// TwinCAT 3 PLC project tcl_AdsObjects
// Title: tcl_AdsObjects
// Company: Red Rock Controls Limited
// Author: R Christopher
// ProjectVersion: 1.1.4.0
// Description: Wrapper classes for Ads function blocks
// ProgramVersion: 3.1.4022.0
// libraries:
//   Tc2_Standard, * (Beckhoff Automation GmbH)
//   Tc2_System, * (Beckhoff Automation GmbH)
//   Tc2_Utilities, * (Beckhoff Automation GmbH)
//   Tc3_Module, * (Beckhoff Automation GmbH)
//   tcl_BaseClasses, * (Red Rock Controls Limited)
//   tcl_UnitTestLibrary, * (Red Rock Controls Limited)
// project tree:
//   / GlobalTextList.TcGTLO
//   POUs/Classes/By Index Group/ T_AdsRead.TcPOU, T_AdsReadWrite.TcPOU, T_AdsWrite.TcPOU
//   POUs/Classes/By Symbol Name/ T_AdsReadBySymbolName.TcPOU, T_AdsReadWriteBySymbolName.TcPOU, T_AdsWriteBySymbolName.TcPOU
//   POUs/Classes/Info/ ST_RawSymbolInfo.TcDUT, T_AdsReadSymbolName.TcPOU, T_AdsReadSymbolInfoByName.TcPOU
//   POUs/Classes/On Change/StructureMonitor/ T_StructureMonitor.TcPOU
//   POUs/Classes/On Change/ T_AdsWriteOnChange.TcPOU
//   Tasks/ PlcTask.TcTTO
//   UnitTests/RPC Example Class/ T_Integer.TcPOU
//   UnitTests/ PB_TestRunner.TcPOU, TestSuite_AdsTests.TcPOU, Test_ReadBySymbolName.TcPOU, Test_ReadBySymbolInfoByName.TcPOU, Test_ReadByIndexGroupAndOffset.TcPOU, Test_ReadSymbolName.TcPOU, Test_ReadBySymbolName_KeepingHandle.TcPOU, Test_ReadWriteBySymbolName.TcPOU, Test_ReadWriteBySymbolName_KeepingHandle.TcPOU, Test_WriteBySymbolName.TcPOU, Test_WriteBySymbolName_KeepingHandle.TcPOU
//   Version/ Global_Version.TcGVL
// real-time tasks:
//   TASK PlcTask: cycle T#10ms, priority 20, ADS port 350

CONFIGURATION tcl_AdsObjects
    RESOURCE PLC ON TwinCAT3
        TASK PlcTask(INTERVAL := T#10ms, PRIORITY := 20);
        PROGRAM PB_TestRunner WITH PlcTask : PB_TestRunner;
    END_RESOURCE
END_CONFIGURATION

// ---- POUs/Classes/Info/ST_RawSymbolInfo.TcDUT
TYPE
    INTERNAL ST_RawSymbolInfo :
    STRUCT
        Address : ULINT;
        Length  : ULINT;
    END_STRUCT
END_TYPE

// ---- Version/Global_Version.TcGVL
{attribute 'TcGenerated'}
{attribute 'no-analysis'}
{attribute 'linkalways'}
// This function has been automatically generated from the project information.
VAR_GLOBAL CONSTANT
	{attribute 'const_non_replaced'}
	stLibVersion_tcl_AdsObjects : ST_LibVersion := (iMajor := 1, iMinor := 1, iBuild := 4, iRevision := 0, nFlags := 1, sVersion := '1.1.4.0');
END_VAR

// ---- UnitTests/PB_TestRunner.TcPOU
PROGRAM PB_TestRunner
VAR
    TestSuite_AdsTests : TestSuite_AdsTests;
END_VAR

TestSuite_AdsTests();

END_PROGRAM

// ---- UnitTests/TestSuite_AdsTests.TcPOU
FUNCTION_BLOCK TestSuite_AdsTests
VAR
    TestRunner : T_TestRunner;
    // Inhibit unused variable warning...                                                        
    {attribute 'analysis' := '-33'} Test_ReadSymbolName                      : Test_ReadSymbolName(TestRunner);
    {attribute 'analysis' := '-33'} Test_ReadBySymbolName                    : Test_ReadBySymbolName(TestRunner);
    {attribute 'analysis' := '-33'} Test_ReadBySymbolName_KeepingHandle      : Test_ReadBySymbolName_KeepingHandle(TestRunner);
    {attribute 'analysis' := '-33'} Test_ReadWriteBySymbolName               : Test_ReadWriteBySymbolName(TestRunner);
    {attribute 'analysis' := '-33'} Test_ReadWriteBySymbolName_KeepingHandle : Test_ReadWriteBySymbolName_KeepingHandle(TestRunner);
    {attribute 'analysis' := '-33'} Test_WriteBySymbolName                   : Test_WriteBySymbolName(TestRunner);
    {attribute 'analysis' := '-33'} Test_WriteBySymbolName_KeepingHandle     : Test_WriteBySymbolName_KeepingHandle(TestRunner);
    {attribute 'analysis' := '-33'} Test_ReadBySymbolInfoByName              : Test_ReadBySymbolInfoByName(TestRunner);
    {attribute 'analysis' := '-33'} Test_ReadByIndexGroupAndOffset           : Test_ReadByIndexGroupAndOffset(TestRunner);

END_VAR

TestRunner(TestSuiteName := 'TestSuite_AdsTests');

END_FUNCTION_BLOCK

// ---- UnitTests/Test_ReadSymbolName.TcPOU
FUNCTION_BLOCK Test_ReadSymbolName EXTENDS T_UnitTestBase
VAR
    AdsPort                                                                                 : UINT;
    AdsReadSymbolName                                                                       : T_AdsReadSymbolName;
    SymbolWithAVeryVeryVeryVeryVeryVeryVeryVeryVeryVeryVeryVeryVeryVeryVeryVeryVeryLongName : INT;
    State                                                                                   : INT;
END_VAR

METHOD Init
State := 0;
END_METHOD

{attribute 'analysis' := '-33'} // inhibit unused variable warning
METHOD RunTest
VAR_OUTPUT
    TestCompleted : BOOL;
    TestFailed    : BOOL;
END_VAR
VAR_INST
    SymbolName : T_MaxString;
END_VAR
CASE State OF
    0:
        AdsPort := _AppInfo.AdsPort;
        AdsReadSymbolName.Execute(Address := ADR(SymbolWithAVeryVeryVeryVeryVeryVeryVeryVeryVeryVeryVeryVeryVeryVeryVeryVeryVeryLongName),
                                  Length  := SIZEOF(SymbolWithAVeryVeryVeryVeryVeryVeryVeryVeryVeryVeryVeryVeryVeryVeryVeryVeryVeryLongName),
                                  PlcPort := AdsPort);
        State := 10;

    10:
        IF NOT AdsReadSymbolName.Execution.Busy THEN
            SymbolName := AdsReadSymbolName.SymbolName;
            State      := 20;
        END_IF

    20:
        AssertTrue(Source    := TestName,
                   Condition := (SymbolName = 'PB_TestRunner.TestSuite_AdsTests.Test_ReadSymbolName.SymbolWithAVeryVeryVeryVeryVeryVeryVeryVeryVeryVeryVeryVeryVeryVeryVeryVeryVeryLongName'),
                   Message   := 'SymbolName read incorrectly',
                   Failed    => TestFailed);

        TestCompleted := TRUE;
END_CASE

AdsReadSymbolName();
END_METHOD

END_FUNCTION_BLOCK

// ---- POUs/Classes/Info/T_AdsReadSymbolName.TcPOU
FUNCTION_BLOCK T_AdsReadSymbolName
VAR
    _Execution    : T_Execution;
    _Address      : PVOID;
    _Length       : UDINT;
    _PlcPort      : UINT;
    _SymbolName   : T_MaxString;
    RawSymbolInfo : ST_RawSymbolInfo;
    AdsRdWrt1     : ADSRDWRTEX;
END_VAR
VAR CONSTANT
    PLCADS_IGR_SYMNAME_BY_ADDR_SIZE : UDINT := 16#40A1;
END_VAR

IF _Execution.Aborting THEN
    _Execution.SetAborted();
END_IF

IF _Execution.Starting THEN
    RawSymbolInfo.Address := _Address;
    RawSymbolInfo.Length  := _Length;
    MEMSET(ADR(_SymbolName), 0, SIZEOF(_SymbolName));
END_IF

AdsRdWrt1(NETID    :=,
          PORT     := _PlcPort,
          IDXGRP   := PLCADS_IGR_SYMNAME_BY_ADDR_SIZE,
          IDXOFFS  := 0,
          WRITELEN := SIZEOF(RawSymbolInfo),
          READLEN  := SIZEOF(SymbolName),
          SRCADDR  := ADR(RawSymbolInfo),
          DESTADDR := ADR(_SymbolName),
          WRTRD    := _Execution.Starting,
          TMOUT    := T#2s,
          BUSY     =>,
          ERR      =>,
          ERRID    =>,
          COUNT_R  =>);

IF _Execution.Starting THEN
    _Execution.SetBusy();
END_IF

IF _Execution.Busy AND NOT AdsRdWrt1.BUSY THEN
    IF AdsRdWrt1.ERR THEN
        _Execution.SetError(F_ErrorIdToString(AdsRdWrt1.ERRID));
    ELSE
        _Execution.SetDone();
    END_IF
END_IF

METHOD Execute : BOOL
VAR_INPUT
    Address : PVOID;
    Length  : UDINT;
    PlcPort : UINT;
END_VAR
THIS^._Address    := Address;
THIS^._Length     := Length;
THIS^._PlcPort    := PlcPort;
THIS^._SymbolName := '';
Execute           := THIS^._Execution.Start();
END_METHOD

PROPERTY Execution : I_Execution
GET
Execution := _Execution;
END_GET
END_PROPERTY

PROPERTY SymbolName : T_MaxString
GET
SymbolName := _SymbolName;
END_GET
END_PROPERTY

END_FUNCTION_BLOCK

// ---- UnitTests/Test_ReadBySymbolName.TcPOU
FUNCTION_BLOCK Test_ReadBySymbolName EXTENDS T_UnitTestBase
VAR
    AdsPort             : UINT;
    AdsReadBySymbolName : T_AdsReadBySymbolName;
    AdsReadSymbolName   : T_AdsReadSymbolName;
    ValueToRead         : INT;
    State               : INT;
END_VAR

METHOD Init
State := 0;
END_METHOD

{attribute 'analysis' := '-33'} // inhibit unused variable warning
METHOD RunTest
VAR_OUTPUT
    TestCompleted : BOOL;
    TestFailed    : BOOL;
END_VAR
VAR_INST
    SymbolName : T_MaxString;
    ReadResult : INT;
END_VAR
CASE State OF
    0:
        AdsPort     := _AppInfo.AdsPort;
        ValueToRead := 1234;
        ReadResult  := 0;
        AdsReadSymbolName.Execute(Address := ADR(ValueToRead),
                                  Length  := SIZEOF(ValueToRead),
                                  PlcPort := AdsPort);
        State := 10;

    10:
        IF NOT AdsReadSymbolName.Execution.Busy THEN
            SymbolName := AdsReadSymbolName.SymbolName;
            State      := 20;
        END_IF

    20:
        AdsReadBySymbolName.Execute(AmsNetId         := '',
                                    Port             := AdsPort,
                                    SymbolName       := SymbolName,
                                    ReadDataAddress  := ADR(ReadResult),
                                    ReadDataLength   := SIZEOF(ReadResult),
                                    KeepSymbolHandle := FALSE);

        State := 30;

    30:
        IF NOT AdsReadBySymbolName.Execution.Busy THEN
            State := 40;
        END_IF

    40:
        AssertTrue(Source    := TestName,
                   Condition := (ReadResult = 1234),
                   Message   := 'Read result <> 1234',
                   Failed    => TestFailed);

        TestCompleted := TRUE;
END_CASE

AdsReadBySymbolName();
AdsReadSymbolName();
END_METHOD

END_FUNCTION_BLOCK

// ---- POUs/Classes/By Symbol Name/T_AdsReadBySymbolName.TcPOU
FUNCTION_BLOCK T_AdsReadBySymbolName
VAR
    _Execution   : T_Execution;
    StateMonitor : T_ValueMonitor;
    State        : INT;

    AmsNetId         : T_AmsNetId;
    Port             : T_AmsPort;
    SymbolName       : T_MaxString;
    ReadDataAddress  : PVOID;
    ReadDataLength   : UDINT;
    KeepSymbolHandle : BOOL;
    SymbolHandle     : DWORD := 0;
    RetryCounter     : T_Counter;

    AdsReadWrite_GetSymHandle : T_AdsReadWrite;
    AdsRead_ReadFromSymbol    : T_AdsRead;
    AdsWrite_ReleaseSymHandle : T_AdsWrite;

END_VAR
VAR CONSTANT
    sInit          : INT := 0;
    sGetHandle     : INT := 1;
    sReadData      : INT := 2;
    sReleaseHandle : INT := 3;
END_VAR

IF _Execution.Aborting THEN
    State := sInit;
    _Execution.SetAborted();
END_IF

StateMonitor.Test(State);
CASE State OF
    sInit:
        IF _Execution.Starting THEN
            _Execution.SetBusy();
            RetryCounter.Reset();
            IF SymbolHandle = 0 THEN
                State := sGetHandle;
            ELSE
                State := sReadData;
            END_IF
        END_IF

    sGetHandle:
        IF StateMonitor.Changed THEN
            // Get a symbol handle from the runtime...
            AdsReadWrite_GetSymHandle.Execute(AmsNetId           := AmsNetId,
                                              Port               := Port,
                                              IndexGroup         := ADSIGRP_SYM_HNDBYNAME,
                                              IndexOffset        := 0,
                                              ArgsAddress        := ADR(SymbolName),
                                              ArgsLength         := INT_TO_UDINT(LEN(SymbolName)),
                                              ReturnValueAddress := ADR(SymbolHandle),
                                              ReturnValueLength  := SIZEOF(SymbolHandle));
        ELSE
            IF AdsReadWrite_GetSymHandle.Execution.Done THEN
                State := sReadData;
            END_IF
            IF AdsReadWrite_GetSymHandle.Execution.Error THEN
                _Execution.SetError(AdsReadWrite_GetSymHandle.Execution.ErrorMsg);
                SymbolHandle := 0;
                State        := sInit;
            END_IF
        END_IF

    sReadData:
        IF StateMonitor.Changed THEN
            // Read the data to from the symbol...
            AdsRead_ReadFromSymbol.Execute(AmsNetId    := AmsNetId,
                                           Port        := Port,
                                           IndexGroup  := ADSIGRP_SYM_VALBYHND,
                                           IndexOffset := SymbolHandle,
                                           DataLength  := ReadDataLength,
                                           DataAddress := ReadDataAddress);
        ELSE
            IF AdsRead_ReadFromSymbol.Execution.Done THEN
                IF KeepSymbolHandle THEN
                    _Execution.SetDone();
                    State := sInit;
                ELSE
                    State := sReleaseHandle;
                END_IF

            ELSIF AdsRead_ReadFromSymbol.Execution.Error THEN
                // Retry if it failed due to an online change invalidating the symbol handle...
                IF RetryCounter.Value = 0 THEN
                    RetryCounter.Inc();
                    SymbolHandle := 0;
                    State        := sGetHandle;
                ELSE
                    _Execution.SetError(AdsRead_ReadFromSymbol.Execution.ErrorMsg);
                    SymbolHandle := 0;
                    State        := sInit;
                END_IF
            END_IF
        END_IF

    sReleaseHandle:
        IF StateMonitor.Changed THEN
            // Release the symbol handle......
            AdsWrite_ReleaseSymHandle.Execute(AmsNetId    := AmsNetId,
                                              Port        := Port,
                                              IndexGroup  := ADSIGRP_SYM_RELEASEHND,
                                              IndexOffset := SymbolHandle,
                                              DataLength  := 0,
                                              DataAddress := 0);
        ELSE
            IF AdsWrite_ReleaseSymHandle.Execution.Done THEN
                // Handle write error to the symbol...
                IF AdsRead_ReadFromSymbol.Execution.Error THEN
                    _Execution.SetError(AdsRead_ReadFromSymbol.Execution.ErrorMsg);
                ELSE
                    _Execution.SetDone();
                END_IF
                SymbolHandle := 0;
                State        := sInit;
            ELSIF AdsWrite_ReleaseSymHandle.Execution.Error THEN
                // Handle release handle error...
                _Execution.SetError(AdsWrite_ReleaseSymHandle.Execution.ErrorMsg);
                SymbolHandle := 0;
                State        := sInit;
            END_IF
        END_IF

END_CASE

AdsReadWrite_GetSymHandle();
AdsRead_ReadFromSymbol();
AdsWrite_ReleaseSymHandle();

METHOD Execute : BOOL
VAR_INPUT
    AmsNetId         : T_AmsNetId;
    Port             : T_AmsPort;
    SymbolName       : T_MaxString;
    ReadDataAddress  : PVOID;
    ReadDataLength   : UDINT;
    KeepSymbolHandle : BOOL;
END_VAR
THIS^.AmsNetId         := AmsNetId;
THIS^.Port             := Port;
THIS^.SymbolName       := SymbolName;
THIS^.ReadDataAddress  := ReadDataAddress;
THIS^.ReadDataLength   := ReadDataLength;
THIS^.KeepSymbolHandle := KeepSymbolHandle;

Execute := _Execution.Start();
END_METHOD

PROPERTY Execution : I_Execution
GET
Execution := _Execution;
END_GET
END_PROPERTY

END_FUNCTION_BLOCK

// ---- POUs/Classes/By Index Group/T_AdsReadWrite.TcPOU
FUNCTION_BLOCK T_AdsReadWrite
VAR_INPUT
END_VAR
VAR_OUTPUT
END_VAR
VAR
    AdsReadWrite : ADSRDWRT;
    _Execution   : T_Execution;
END_VAR

IF _Execution.Aborting THEN
    _Execution.SetAborted();
END_IF

AdsReadWrite(NETID    :=,
             PORT     :=,
             IDXGRP   :=,
             IDXOFFS  :=,
             WRITELEN :=,
             READLEN  :=,
             SRCADDR  :=,
             DESTADDR :=,
             WRTRD    := _Execution.Starting,
             TMOUT    :=,
             BUSY     =>,
             ERR      =>,
             ERRID    =>);

IF _Execution.Starting THEN
    _Execution.SetBusy();
END_IF
IF _Execution.Busy AND NOT AdsReadWrite.BUSY THEN
    IF AdsReadWrite.ERR THEN
        _Execution.SetError(F_ErrorIdToString(AdsReadWrite.ERRID));
    ELSE
        _Execution.SetDone();
    END_IF
END_IF

METHOD Execute : BOOL
VAR_INPUT
    AmsNetId           : T_AmsNetID;
    Port               : T_AmsPort;
    IndexGroup         : UDINT;
    IndexOffset        : UDINT;
    ArgsAddress        : PVOID;
    ArgsLength         : UDINT;
    ReturnValueAddress : PVOID;
    ReturnValueLength  : UDINT;
END_VAR
IF _Execution.Start() THEN
    AdsReadWrite.NETID   := AmsNetId;
    AdsReadWrite.PORT    := Port;
    AdsReadWrite.IDXGRP  := IndexGroup;
    AdsReadWrite.IDXOFFS := IndexOffset;
    // Data to be written...
    AdsReadWrite.SRCADDR  := ArgsAddress;
    AdsReadWrite.WRITELEN := ArgsLength;
    // Data returned...
    AdsReadWrite.DESTADDR := ReturnValueAddress;
    AdsReadWrite.READLEN  := ReturnValueLength;
END_IF
END_METHOD

PROPERTY Execution : I_Execution
GET
Execution := _Execution;
END_GET
END_PROPERTY

END_FUNCTION_BLOCK

// ---- POUs/Classes/By Index Group/T_AdsRead.TcPOU
FUNCTION_BLOCK T_AdsRead
VAR
    _Execution : T_Execution;
    AdsRead1   : ADSREAD := (TMOUT := T#2S);
END_VAR

IF _Execution.Aborting THEN
    _Execution.SetAborted();
END_IF

AdsRead1(NETID    :=,
         PORT     :=,
         IDXGRP   :=,
         IDXOFFS  :=,
         LEN      :=,
         DESTADDR :=,
         READ     := _Execution.Starting,
         TMOUT    :=,
         BUSY     =>,
         ERR      =>,
         ERRID    =>);

IF _Execution.Starting THEN
    _Execution.SetBusy();
END_IF
IF _Execution.Busy AND NOT AdsRead1.BUSY THEN
    IF AdsRead1.ERR THEN
        _Execution.SetError(F_ErrorIdToString(AdsRead1.ERRID));
    ELSE
        _Execution.SetDone();
    END_IF
END_IF

METHOD Execute : BOOL
VAR_INPUT
    AmsNetId    : T_AmsNetid;
    Port        : T_AmsPort;
    IndexGroup  : UDINT;
    IndexOffset : UDINT;
    DataLength  : UDINT;
    DataAddress : PVOID;
END_VAR
AdsRead1.NETID    := AmsNetId;
AdsRead1.PORT     := Port;
AdsRead1.IDXGRP   := IndexGroup;
AdsRead1.IDXOFFS  := IndexOffset;
AdsRead1.LEN      := DataLength;
AdsRead1.DESTADDR := DataAddress;

Execute := _Execution.Start();
END_METHOD

PROPERTY Execution : I_Execution
GET
Execution := _Execution;
END_GET
END_PROPERTY

END_FUNCTION_BLOCK

// ---- POUs/Classes/By Index Group/T_AdsWrite.TcPOU
FUNCTION_BLOCK T_AdsWrite
VAR
    _Execution : T_Execution;
    AdsWrite1  : ADSWRITE := (TMOUT := T#2S);
END_VAR

IF _Execution.Aborting THEN
    _Execution.SetAborted();
END_IF

AdsWrite1(NETID   :=,
          PORT    :=,
          IDXGRP  :=,
          IDXOFFS :=,
          LEN     :=,
          SRCADDR :=,
          WRITE   := _Execution.Starting,
          TMOUT   :=,
          BUSY    =>,
          ERR     =>,
          ERRID   =>);

IF _Execution.Starting THEN
    _Execution.SetBusy();
END_IF
IF _Execution.Busy AND NOT AdsWrite1.BUSY THEN
    IF AdsWrite1.ERR THEN
        _Execution.SetError(F_ErrorIdToString(AdsWrite1.ERRID));
    ELSE
        _Execution.SetDone();
    END_IF
END_IF

METHOD Execute : BOOL
VAR_INPUT
    AmsNetId    : T_AmsNetid;
    Port        : T_AmsPort;
    IndexGroup  : UDINT;
    IndexOffset : UDINT;
    DataLength  : UDINT;
    DataAddress : PVOID;
END_VAR
AdsWrite1.NETID   := AmsNetId;
AdsWrite1.PORT    := Port;
AdsWrite1.IDXGRP  := IndexGroup;
AdsWrite1.IDXOFFS := IndexOffset;
AdsWrite1.LEN     := DataLength;
AdsWrite1.SRCADDR := DataAddress;
Execute           := _Execution.Start();
END_METHOD

PROPERTY Execution : I_Execution
GET
Execution := _Execution;
END_GET
END_PROPERTY

END_FUNCTION_BLOCK

// ---- UnitTests/Test_ReadBySymbolName_KeepingHandle.TcPOU
FUNCTION_BLOCK Test_ReadBySymbolName_KeepingHandle EXTENDS T_UnitTestBase
VAR
    AdsPort             : UINT;
    AdsReadBySymbolName : T_AdsReadBySymbolName;
    AdsReadSymbolName   : T_AdsReadSymbolName;
    ValueToRead         : INT;
    State               : INT;
END_VAR

METHOD Init
State := 0;
END_METHOD

{attribute 'analysis' := '-33'} // inhibit unused variable warning
METHOD RunTest
VAR_OUTPUT
    TestCompleted : BOOL;
    TestFailed    : BOOL;
END_VAR
VAR_INST
    SymbolName : T_MaxString;
    ReadResult : INT;
END_VAR
CASE State OF
    0:
        AdsPort     := _AppInfo.AdsPort;
        ValueToRead := 1234;
        ReadResult  := 0;
        AdsReadSymbolName.Execute(Address := ADR(ValueToRead),
                                  Length  := SIZEOF(ValueToRead),
                                  PlcPort := AdsPort);
        State := 10;

    10:
        IF NOT AdsReadSymbolName.Execution.Busy THEN
            SymbolName := AdsReadSymbolName.SymbolName;
            State      := 20;
        END_IF

    20:
        AdsReadBySymbolName.Execute(AmsNetId         := '',
                                    Port             := AdsPort,
                                    SymbolName       := SymbolName,
                                    ReadDataAddress  := ADR(ReadResult),
                                    ReadDataLength   := SIZEOF(ReadResult),
                                    KeepSymbolHandle := TRUE);

        State := 30;

    30:
        IF NOT AdsReadBySymbolName.Execution.Busy THEN
            State := 40;
        END_IF

    40:
        AssertTrue(Source    := TestName,
                   Condition := (ReadResult = 1234),
                   Message   := 'Read result <> 1234',
                   Failed    => TestFailed);
        IF TestFailed THEN
            TestCompleted := TRUE;
        ELSE
            State := 50;
        END_IF

    50:
        AssertTrue(Source    := TestName,
                   Condition := (AdsReadBySymbolName.SymbolHandle <> 0),
                   Message   := 'SymbolHandle was released',
                   Failed    => TestFailed);

        TestCompleted := TRUE;
END_CASE

AdsReadBySymbolName();
AdsReadSymbolName();
END_METHOD

END_FUNCTION_BLOCK

// ---- UnitTests/Test_ReadWriteBySymbolName.TcPOU
FUNCTION_BLOCK Test_ReadWriteBySymbolName EXTENDS T_UnitTestBase
VAR
    AdsPort                  : UINT;
    AdsReadWriteBySymbolName : T_AdsReadWriteBySymbolName;
    AdsReadSymbolName        : T_AdsReadSymbolName;
    TestInteger              : T_Integer;
    State                    : INT;
END_VAR

METHOD Init
State := 0;
END_METHOD

{attribute 'analysis' := '-33'} // inhibit unused variable warning
METHOD RunTest
VAR_OUTPUT
    TestCompleted : BOOL;
    TestFailed    : BOOL;
END_VAR
VAR_INST
    SymbolName      : T_MaxString;
    ReadWriteResult : INT;
END_VAR
CASE State OF
    0:
        AdsPort := _AppInfo.AdsPort;
        TestInteger.Init(1111);
        ReadWriteResult := 0;
        AdsReadSymbolName.Execute(Address := ADR(TestInteger),
                                  Length  := SIZEOF(TestInteger),
                                  PlcPort := AdsPort);
        State := 10;

    10:
        IF NOT AdsReadSymbolName.Execution.Busy THEN
            SymbolName := CONCAT(AdsReadSymbolName.SymbolName, '#Inc');
            State      := 20;
        END_IF

    20:
        AdsReadWriteBySymbolName.Execute(AmsNetId         := '',
                                         Port             := AdsPort,
                                         SymbolName       := SymbolName,
                                         ReadDataAddress  := ADR(ReadWriteResult),
                                         ReadDataLength   := SIZEOF(ReadWriteResult),
                                         WriteDataAddress := 0,
                                         WriteDataLength  := 0,
                                         KeepSymbolHandle := FALSE);

        State := 30;

    30:
        IF NOT AdsReadWriteBySymbolName.Execution.Busy THEN
            State := 40;
        END_IF

    40:
        AssertTrue(Source    := TestName,
                   Condition := (ReadWriteResult = 1112),
                   Message   := 'ReadWriteResult <> 1112',
                   Failed    => TestFailed);

        TestCompleted := TRUE;
END_CASE

AdsReadWriteBySymbolName();
AdsReadSymbolName();
END_METHOD

END_FUNCTION_BLOCK

// ---- POUs/Classes/By Symbol Name/T_AdsReadWriteBySymbolName.TcPOU
FUNCTION_BLOCK T_AdsReadWriteBySymbolName
VAR
    _Execution   : T_Execution;
    StateMonitor : T_ValueMonitor;
    State        : INT;

    AmsNetId         : T_AmsNetId;
    Port             : T_AmsPort;
    SymbolName       : T_MaxString;
    ReadDataAddress  : PVOID;
    ReadDataLength   : UDINT;
    WriteDataAddress : PVOID;
    WriteDataLength  : UDINT;
    KeepSymbolHandle : BOOL;
    SymbolHandle     : DWORD := 0;
    RetryCounter     : T_Counter;

    AdsReadWrite_GetSymHandle : T_AdsReadWrite;
    AdsReadWrite_ToSymbol     : T_AdsReadWrite;
    AdsWrite_ReleaseSymHandle : T_AdsWrite;

END_VAR
VAR CONSTANT
    sInit          : INT := 0;
    sGetHandle     : INT := 1;
    sReadWrite     : INT := 2;
    sReleaseHandle : INT := 3;
END_VAR

IF _Execution.Aborting THEN
    State := sInit;
    _Execution.SetAborted();
END_IF

StateMonitor.Test(State);
CASE State OF
    sInit:
        IF _Execution.Starting THEN
            _Execution.SetBusy();
            RetryCounter.Reset();
            IF SymbolHandle = 0 THEN
                State := sGetHandle;
            ELSE
                State := sReadWrite;
            END_IF
        END_IF

    sGetHandle:
        IF StateMonitor.Changed THEN
            // Get a symbol handle from the runtime...
            AdsReadWrite_GetSymHandle.Execute(AmsNetId           := AmsNetId,
                                              Port               := Port,
                                              IndexGroup         := ADSIGRP_SYM_HNDBYNAME,
                                              IndexOffset        := 0,
                                              ArgsAddress        := ADR(SymbolName),
                                              ArgsLength         := INT_TO_UDINT(LEN(SymbolName)),
                                              ReturnValueAddress := ADR(SymbolHandle),
                                              ReturnValueLength  := SIZEOF(SymbolHandle));
        ELSE
            IF AdsReadWrite_GetSymHandle.Execution.Done THEN
                State := sReadWrite;
            END_IF
            IF AdsReadWrite_GetSymHandle.Execution.Error THEN
                _Execution.SetError(AdsReadWrite_GetSymHandle.Execution.ErrorMsg);
                SymbolHandle := 0;
                State        := sInit;
            END_IF
        END_IF

    sReadWrite:
        IF StateMonitor.Changed THEN
            // Write the data to the symbol...
            AdsReadWrite_ToSymbol.Execute(AmsNetId           := AmsNetId,
                                          Port               := Port,
                                          IndexGroup         := ADSIGRP_SYM_VALBYHND,
                                          IndexOffset        := SymbolHandle,
                                          ArgsAddress        := WriteDataAddress,
                                          ArgsLength         := WriteDataLength,
                                          ReturnValueAddress := ReadDataAddress,
                                          ReturnValueLength  := ReadDataLength);

        ELSE
            IF AdsReadWrite_ToSymbol.Execution.Done THEN
                IF KeepSymbolHandle THEN
                    _Execution.SetDone();
                    State := sInit;
                ELSE
                    State := sReleaseHandle;
                END_IF

            ELSIF AdsReadWrite_ToSymbol.Execution.Error THEN
                // Retry if it failed due to an online change invalidating the symbol handle...
                IF RetryCounter.Value = 0 THEN
                    RetryCounter.Inc();
                    SymbolHandle := 0;
                    State        := sGetHandle;
                ELSE
                    _Execution.SetError(AdsReadWrite_ToSymbol.Execution.ErrorMsg);
                    SymbolHandle := 0;
                    State        := sInit;
                END_IF
            END_IF
        END_IF

    sReleaseHandle:
        IF StateMonitor.Changed THEN
            // Release the symbol handle......
            AdsWrite_ReleaseSymHandle.Execute(AmsNetId    := AmsNetId,
                                              Port        := Port,
                                              IndexGroup  := ADSIGRP_SYM_RELEASEHND,
                                              IndexOffset := SymbolHandle,
                                              DataLength  := 0,
                                              DataAddress := 0);
        ELSE
            IF AdsWrite_ReleaseSymHandle.Execution.Done THEN
                // Handle write error to the symbol...
                IF AdsReadWrite_ToSymbol.Execution.Error THEN
                    _Execution.SetError(AdsReadWrite_ToSymbol.Execution.ErrorMsg);
                ELSE
                    _Execution.SetDone();
                END_IF
                SymbolHandle := 0;
                State        := sInit;
            ELSIF AdsWrite_ReleaseSymHandle.Execution.Error THEN
                // Handle release handle error...
                _Execution.SetError(AdsWrite_ReleaseSymHandle.Execution.ErrorMsg);
                SymbolHandle := 0;
                State        := sInit;
            END_IF
        END_IF

END_CASE

AdsReadWrite_GetSymHandle();
AdsReadWrite_ToSymbol();
AdsWrite_ReleaseSymHandle();

METHOD Execute : BOOL
VAR_INPUT
    AmsNetId         : T_AmsNetId;
    Port             : T_AmsPort;
    SymbolName       : T_MaxString;
    ReadDataAddress  : PVOID;
    ReadDataLength   : UDINT;
    WriteDataAddress : PVOID;
    WriteDataLength  : UDINT;
    KeepSymbolHandle : BOOL;
END_VAR
THIS^.AmsNetId         := AmsNetId;
THIS^.Port             := Port;
THIS^.SymbolName       := SymbolName;
THIS^.ReadDataAddress  := ReadDataAddress;
THIS^.ReadDataLength   := ReadDataLength;
THIS^.WriteDataAddress := WriteDataAddress;
THIS^.WriteDataLength  := WriteDataLength;
THIS^.KeepSymbolHandle := KeepSymbolHandle;

Execute := _Execution.Start();
END_METHOD

PROPERTY Execution : I_Execution
GET
Execution := _Execution;
END_GET
END_PROPERTY

END_FUNCTION_BLOCK

// ---- UnitTests/RPC Example Class/T_Integer.TcPOU
{attribute 'hide'}
{attribute 'reflection'}
FUNCTION_BLOCK T_Integer
VAR
    Value : INT;
END_VAR

{attribute 'TcRpcEnable'}
METHOD Inc : INT
VAR_INPUT
END_VAR
Value := Value + 1;
Inc   := Value;
END_METHOD

METHOD Init
VAR_INPUT
    Value : INT;
END_VAR
THIS^.Value := Value;
END_METHOD

END_FUNCTION_BLOCK

// ---- UnitTests/Test_ReadWriteBySymbolName_KeepingHandle.TcPOU
FUNCTION_BLOCK Test_ReadWriteBySymbolName_KeepingHandle EXTENDS T_UnitTestBase
VAR
    AdsPort                  : UINT;
    AdsReadWriteBySymbolName : T_AdsReadWriteBySymbolName;
    AdsReadSymbolName        : T_AdsReadSymbolName;
    TestInteger              : T_Integer;
    State                    : INT;
END_VAR

METHOD Init
State := 0;
END_METHOD

{attribute 'analysis' := '-33'} // inhibit unused variable warning
METHOD RunTest
VAR_OUTPUT
    TestCompleted : BOOL;
    TestFailed    : BOOL;
END_VAR
VAR_INST
    SymbolName      : T_MaxString;
    ReadWriteResult : INT;
END_VAR
CASE State OF
    0:
        AdsPort := _AppInfo.AdsPort;
        TestInteger.Init(1111);
        ReadWriteResult := 0;
        AdsReadSymbolName.Execute(Address := ADR(TestInteger),
                                  Length  := SIZEOF(TestInteger),
                                  PlcPort := AdsPort);
        State := 10;

    10:
        IF NOT AdsReadSymbolName.Execution.Busy THEN
            SymbolName := CONCAT(AdsReadSymbolName.SymbolName, '#Inc');
            State      := 20;
        END_IF

    20:
        AdsReadWriteBySymbolName.Execute(AmsNetId         := '',
                                         Port             := AdsPort,
                                         SymbolName       := SymbolName,
                                         ReadDataAddress  := ADR(ReadWriteResult),
                                         ReadDataLength   := SIZEOF(ReadWriteResult),
                                         WriteDataAddress := 0,
                                         WriteDataLength  := 0,
                                         KeepSymbolHandle := FALSE);

        State := 30;

    30:
        IF NOT AdsReadWriteBySymbolName.Execution.Busy THEN
            State := 40;
        END_IF

    40:
        AssertTrue(Source    := TestName,
                   Condition := (ReadWriteResult = 1112),
                   Message   := 'ReadWriteResult <> 1112',
                   Failed    => TestFailed);

        TestCompleted := TRUE;
END_CASE

AdsReadWriteBySymbolName();
AdsReadSymbolName();
END_METHOD

END_FUNCTION_BLOCK

// ---- UnitTests/Test_WriteBySymbolName.TcPOU
FUNCTION_BLOCK Test_WriteBySymbolName EXTENDS T_UnitTestBase
VAR
    AdsPort              : UINT;
    AdsWriteBySymbolName : T_AdsWriteBySymbolName;
    AdsReadSymbolName    : T_AdsReadSymbolName;
    WriteResult          : INT; // We are writing to this variable by its symbol name
    State                : INT;
END_VAR

METHOD Init
State := 0;
END_METHOD

{attribute 'analysis' := '-33'} // inhibit unused variable warning
METHOD RunTest
VAR_OUTPUT
    TestCompleted : BOOL;
    TestFailed    : BOOL;
END_VAR
VAR_INST
    SymbolName   : T_MaxString;
    ValueToWrite : INT;
END_VAR
CASE State OF
    0:
        AdsPort      := _AppInfo.AdsPort;
        ValueToWrite := 3456;
        WriteResult  := 0;
        AdsReadSymbolName.Execute(Address := ADR(WriteResult),
                                  Length  := SIZEOF(WriteResult),
                                  PlcPort := AdsPort);
        State := 10;

    10:
        IF NOT AdsReadSymbolName.Execution.Busy THEN
            SymbolName := AdsReadSymbolName.SymbolName;
            State      := 20;
        END_IF

    20:
        AdsWriteBySymbolName.Execute(AmsNetId         := '',
                                     Port             := AdsPort,
                                     SymbolName       := SymbolName,
                                     WriteDataAddress := ADR(ValueToWrite),
                                     WriteDataLength  := SIZEOF(ValueToWrite),
                                     KeepSymbolHandle := FALSE);

        State := 30;

    30:
        IF NOT AdsWriteBySymbolName.Execution.Busy THEN
            State := 40;
        END_IF

    40:
        AssertTrue(Source    := TestName,
                   Condition := (WriteResult = 3456),
                   Message   := 'WriteResult <> 3456',
                   Failed    => TestFailed);

        TestCompleted := TRUE;
END_CASE

AdsWriteBySymbolName();
AdsReadSymbolName();
END_METHOD

END_FUNCTION_BLOCK

// ---- POUs/Classes/By Symbol Name/T_AdsWriteBySymbolName.TcPOU
FUNCTION_BLOCK T_AdsWriteBySymbolName
VAR
    _Execution   : T_Execution;
    StateMonitor : T_ValueMonitor;
    State        : INT;

    AmsNetId         : T_AmsNetId;
    Port             : T_AmsPort;
    SymbolName       : T_MaxString; // Symbol name of variable to write to
    WriteDataAddress : PVOID;       // Address of data to write
    WriteDataLength  : UDINT;       // Sizeof data to write
    KeepSymbolHandle : BOOL;        // Handle is not released after writing - useful for multiple writes to the same symbol
    SymbolHandle     : DWORD := 0;
    RetryCounter     : T_Counter;

    AdsReadWrite_GetSymHandle : T_AdsReadWrite;
    AdsWrite_WriteToSymbol    : T_AdsWrite;
    AdsWrite_ReleaseSymHandle : T_AdsWrite;
END_VAR
VAR CONSTANT
    sInit          : INT := 0;
    sGetHandle     : INT := 1;
    sWriteData     : INT := 2;
    sReleaseHandle : INT := 3;
END_VAR

IF _Execution.Aborting THEN
    State := sInit;
    _Execution.SetAborted();
END_IF

StateMonitor.Test(State);
CASE State OF
    sInit:
        IF _Execution.Starting THEN
            _Execution.SetBusy();
            RetryCounter.Reset();
            IF SymbolHandle = 0 THEN
                State := sGetHandle;
            ELSE
                State := sWriteData;
            END_IF
        END_IF

    sGetHandle:
        IF StateMonitor.Changed THEN
            // Get a symbol handle from the runtime...
            AdsReadWrite_GetSymHandle.Execute(AmsNetId           := AmsNetId,
                                              Port               := Port,
                                              IndexGroup         := ADSIGRP_SYM_HNDBYNAME,
                                              IndexOffset        := 0,
                                              ArgsAddress        := ADR(SymbolName),
                                              ArgsLength         := INT_TO_UDINT(LEN(SymbolName)),
                                              ReturnValueAddress := ADR(SymbolHandle),
                                              ReturnValueLength  := SIZEOF(SymbolHandle));
        ELSE
            IF AdsReadWrite_GetSymHandle.Execution.Done THEN
                State := sWriteData;
            END_IF
            IF AdsReadWrite_GetSymHandle.Execution.Error THEN
                _Execution.SetError(AdsReadWrite_GetSymHandle.Execution.ErrorMsg);
                SymbolHandle := 0;
                State        := sInit;
            END_IF
        END_IF

    sWriteData:
        IF StateMonitor.Changed THEN
            // Write the data to the symbol...
            AdsWrite_WriteToSymbol.Execute(AmsNetId    := AmsNetId,
                                           Port        := Port,
                                           IndexGroup  := ADSIGRP_SYM_VALBYHND,
                                           IndexOffset := SymbolHandle,
                                           DataLength  := WriteDataLength,
                                           DataAddress := WriteDataAddress);
        ELSE
            IF AdsWrite_WriteToSymbol.Execution.Done THEN
                IF KeepSymbolHandle THEN
                    _Execution.SetDone();
                    State := sInit;
                ELSE
                    State := sReleaseHandle;
                END_IF

            ELSIF AdsWrite_WriteToSymbol.Execution.Error THEN
                // Retry if it failed due to an online change invalidating the symbol handle...
                IF RetryCounter.Value = 0 THEN
                    RetryCounter.Inc();
                    SymbolHandle := 0;
                    State        := sGetHandle;
                ELSE
                    _Execution.SetError(AdsWrite_WriteToSymbol.Execution.ErrorMsg);
                    SymbolHandle := 0;
                    State        := sInit;
                END_IF
            END_IF
        END_IF

    sReleaseHandle:
        IF StateMonitor.Changed THEN
            // Release the symbol handle......
            AdsWrite_ReleaseSymHandle.Execute(AmsNetId    := AmsNetId,
                                              Port        := Port,
                                              IndexGroup  := ADSIGRP_SYM_RELEASEHND,
                                              IndexOffset := SymbolHandle,
                                              DataLength  := 0,
                                              DataAddress := 0);
        ELSE
            IF AdsWrite_ReleaseSymHandle.Execution.Done THEN
                // Handle write error to the symbol...
                IF AdsWrite_WriteToSymbol.Execution.Error THEN
                    _Execution.SetError(AdsWrite_WriteToSymbol.Execution.ErrorMsg);
                ELSE
                    _Execution.SetDone();
                END_IF
                SymbolHandle := 0;
                State        := sInit;
            ELSIF AdsWrite_ReleaseSymHandle.Execution.Error THEN
                // Handle release handle error...
                _Execution.SetError(AdsWrite_ReleaseSymHandle.Execution.ErrorMsg);
                SymbolHandle := 0;
                State        := sInit;
            ELSIF AdsWrite_WriteToSymbol.Execution.Error THEN
                // Handle Write To Symbol error...
                _Execution.SetError(AdsWrite_WriteToSymbol.Execution.ErrorMsg);
                SymbolHandle := 0;
                State        := sInit;
            END_IF
        END_IF

END_CASE

AdsReadWrite_GetSymHandle();
AdsWrite_WriteToSymbol();
AdsWrite_ReleaseSymHandle();

METHOD Execute : BOOL
VAR_INPUT
    AmsNetId         : T_AmsNetId;  // of Machine to write to
    Port             : T_AmsPort;   // of PLC to write to
    SymbolName       : T_MaxString; // of variable to write to                                                 
    WriteDataAddress : PVOID;       // of data to write                                                            
    WriteDataLength  : UDINT;       // of data to write                                                                
    KeepSymbolHandle : BOOL;        // Handle is not released after writing - useful for multiple writes to the same symbol
END_VAR
THIS^.AmsNetId         := AmsNetId;
THIS^.Port             := Port;
THIS^.SymbolName       := SymbolName;
THIS^.WriteDataAddress := WriteDataAddress;
THIS^.WriteDataLength  := WriteDataLength;
THIS^.KeepSymbolHandle := KeepSymbolHandle;

Execute := _Execution.Start();
END_METHOD

PROPERTY Execution : I_Execution
GET
Execution := _Execution;
END_GET
END_PROPERTY

END_FUNCTION_BLOCK

// ---- UnitTests/Test_WriteBySymbolName_KeepingHandle.TcPOU
FUNCTION_BLOCK Test_WriteBySymbolName_KeepingHandle EXTENDS T_UnitTestBase
VAR
    AdsPort              : UINT;
    AdsWriteBySymbolName : T_AdsWriteBySymbolName;
    AdsReadSymbolName    : T_AdsReadSymbolName;
    WriteResult          : INT; // We are writing to this variable by its symbol name
    State                : INT;
END_VAR

METHOD Init
State := 0;
END_METHOD

{attribute 'analysis' := '-33'} // inhibit unused variable warning
METHOD RunTest
VAR_OUTPUT
    TestCompleted : BOOL;
    TestFailed    : BOOL;
END_VAR
VAR_INST
    SymbolName   : T_MaxString;
    ValueToWrite : INT;
END_VAR
CASE State OF
    0:
        AdsPort      := _AppInfo.AdsPort;
        ValueToWrite := 3456;
        WriteResult  := 0;
        AdsReadSymbolName.Execute(Address := ADR(WriteResult),
                                  Length  := SIZEOF(WriteResult),
                                  PlcPort := AdsPort);
        State := 10;

    10:
        IF NOT AdsReadSymbolName.Execution.Busy THEN
            SymbolName := AdsReadSymbolName.SymbolName;
            State      := 20;
        END_IF

    20:
        AdsWriteBySymbolName.Execute(AmsNetId         := '',
                                     Port             := AdsPort,
                                     SymbolName       := SymbolName,
                                     WriteDataAddress := ADR(ValueToWrite),
                                     WriteDataLength  := SIZEOF(ValueToWrite),
                                     KeepSymbolHandle := TRUE);

        State := 30;

    30:
        IF NOT AdsWriteBySymbolName.Execution.Busy THEN
            State := 40;
        END_IF

    40:
        AssertTrue(Source    := TestName,
                   Condition := (WriteResult = 3456),
                   Message   := 'WriteResult <> 3456',
                   Failed    => TestFailed);

        TestCompleted := TRUE;
END_CASE

AdsWriteBySymbolName();
AdsReadSymbolName();
END_METHOD

END_FUNCTION_BLOCK

// ---- UnitTests/Test_ReadBySymbolInfoByName.TcPOU
FUNCTION_BLOCK Test_ReadBySymbolInfoByName EXTENDS T_UnitTestBase
VAR
    AdsPort                 : UINT;
    AdsReadSymbolInfoByName : T_AdsReadSymbolInfoByName;
    AdsReadSymbolName       : T_AdsReadSymbolName;
    SymbolUnderTest         : LREAL; // Comment describing Symbol
    State                   : INT;
END_VAR

METHOD Init
State := 0;
END_METHOD

{attribute 'analysis' := '-33'} // inhibit unused variable warning
METHOD RunTest
VAR_OUTPUT
    TestCompleted : BOOL;
    TestFailed    : BOOL;
END_VAR
VAR_INST
    SymbolName : T_MaxString;
    ReadResult : INT;
    SymbolInfo : SYMINFOSTRUCT;
END_VAR
CASE State OF
    0:
        AdsPort    := _AppInfo.AdsPort;
        ReadResult := 0;
        AdsReadSymbolName.Execute(Address := ADR(SymbolUnderTest),
                                  Length  := SIZEOF(SymbolUnderTest),
                                  PlcPort := AdsPort);
        State := 10;

    10:
        IF NOT AdsReadSymbolName.Execution.Busy THEN
            SymbolName := AdsReadSymbolName.SymbolName;
            State      := 20;
        END_IF

    20:
        AdsReadSymbolInfoByName.Execute(SymbolName := SymbolName,
                                        PlcPort    := AdsPort);

        State := 30;

    30:
        IF NOT AdsReadSymbolInfoByName.Execution.Busy THEN
            SymbolInfo := AdsReadSymbolInfoByName.SymbolInfo;
            State      := 40;
        END_IF

    40:
        AssertTrue(Source    := TestName,
                   Condition := SymbolInfo.adsDataType = ADSDATATYPEID.ADST_REAL64,
                   Message   := 'adsDataType not correct',
                   Failed    => TestFailed);
        IF TestFailed THEN
            TestCompleted := TRUE;
            RETURN;
        END_IF

        AssertTrue(Source    := TestName,
                   Condition := SymbolInfo.byteSize = 8,
                   Message   := 'byteSize not correct',
                   Failed    => TestFailed);
        IF TestFailed THEN
            TestCompleted := TRUE;
            RETURN;
        END_IF

        AssertTrue(Source    := TestName,
                   Condition := SymbolInfo.symDataType = 'LREAL',
                   Message   := 'symDataType not correct',
                   Failed    => TestFailed);
        IF TestFailed THEN
            TestCompleted := TRUE;
            RETURN;
        END_IF

        AssertTrue(Source    := TestName,
                   Condition := SymbolInfo.symComment = ' Comment describing Symbol',
                   Message   := 'symComment not correct',
                   Failed    => TestFailed);
        IF TestFailed THEN
            TestCompleted := TRUE;
            RETURN;
        END_IF

        TestCompleted := TRUE;
END_CASE

AdsReadSymbolInfoByName();
AdsReadSymbolName();
END_METHOD

END_FUNCTION_BLOCK

// ---- POUs/Classes/Info/T_AdsReadSymbolInfoByName.TcPOU
FUNCTION_BLOCK T_AdsReadSymbolInfoByName
VAR
    _Execution             : T_Execution;
    PLC_ReadSymInfoByName1 : PLC_ReadSymInfoByName;
END_VAR

IF _Execution.Aborting THEN
    _Execution.SetAborted();
END_IF

PLC_ReadSymInfoByName1(NETID   := '',
                       PORT    :=,
                       SYMNAME :=,
                       START   := _Execution.Starting,
                       TMOUT   := T#2S,
                       BUSY    =>,
                       ERR     =>,
                       ERRID   =>,
                       SYMINFO =>);

IF _Execution.Starting THEN
    _Execution.SetBusy();
END_IF

IF _Execution.Busy AND NOT PLC_ReadSymInfoByName1.BUSY THEN
    IF PLC_ReadSymInfoByName1.ERR THEN
        _Execution.SetError(F_ErrorIdToString(PLC_ReadSymInfoByName1.ERRID));
    ELSE
        _Execution.SetDone();
    END_IF
END_IF

METHOD Execute : BOOL
VAR_INPUT
    SymbolName : T_MaxString;
    PlcPort    : UINT;
END_VAR
PLC_ReadSymInfoByName1.SYMNAME := SymbolName;
PLC_ReadSymInfoByName1.PORT    := PlcPort;
Execute                        := THIS^._Execution.Start();
END_METHOD

PROPERTY Execution : I_Execution
GET
Execution := _Execution;
END_GET
END_PROPERTY

PROPERTY SymbolInfo : REFERENCE TO SYMINFOSTRUCT
GET
SymbolInfo REF= PLC_ReadSymInfoByName1.SYMINFO;
END_GET
END_PROPERTY

END_FUNCTION_BLOCK

// ---- UnitTests/Test_ReadByIndexGroupAndOffset.TcPOU
FUNCTION_BLOCK Test_ReadByIndexGroupAndOffset EXTENDS T_UnitTestBase
VAR
    AdsPort               : UINT;
    AdsRead               : T_AdsRead;
    ValueToRead AT %MB100 : INT;
    State                 : INT;
END_VAR

METHOD Init
State := 0;
END_METHOD

{attribute 'analysis' := '-33'} // inhibit unused variable warning
METHOD RunTest
VAR_OUTPUT
    TestCompleted : BOOL;
    TestFailed    : BOOL;
END_VAR
VAR_INST
    SymbolName : T_MaxString;
    ReadResult : INT;
END_VAR
CASE State OF
    0:
        AdsPort     := _AppInfo.AdsPort;
        ValueToRead := 1234;
        ReadResult  := 0;
        AdsRead.Execute(AmsNetId    := '',
                        Port        := AdsPort,
                        IndexGroup  := 16#4020,
                        IndexOffset := 100,
                        DataLength  := SIZEOF(ReadResult),
                        DataAddress := ADR(ReadResult));

        State := 10;

    10:
        IF NOT AdsRead.Execution.Busy THEN
            State := 20;
        END_IF

    20:
        AssertTrue(Source    := TestName,
                   Condition := (ReadResult = 1234),
                   Message   := 'Read result <> 1234',
                   Failed    => TestFailed);

        TestCompleted := TRUE;
END_CASE

AdsRead();
END_METHOD

END_FUNCTION_BLOCK

// ---- POUs/Classes/On Change/StructureMonitor/T_StructureMonitor.TcPOU
{attribute 'no_explicit_call':= 'do not call this POU directly'}
FUNCTION_BLOCK T_StructureMonitor
VAR
    _Changed   : BOOL;
    Stored_CRC : WORD := 16#FFFF;
END_VAR

PROPERTY Changed : BOOL
GET
Changed := _Changed;
END_GET
END_PROPERTY

METHOD Reset
VAR_INPUT
END_VAR
Stored_CRC := 16#FFFF;
END_METHOD

METHOD Test
VAR_INPUT
    StructureAddress : POINTER TO BYTE;
    StructureSize    : UDINT;
END_VAR
VAR
    CRC : WORD;
END_VAR
CRC := F_DATA_TO_CRC16_CCITT(pData  := StructureAddress,
                             cbData := StructureSize,
                             crc    := 0);

_Changed := (CRC <> Stored_CRC);

IF Changed THEN
    Stored_CRC := CRC;
END_IF
END_METHOD

END_FUNCTION_BLOCK

// ---- POUs/Classes/On Change/T_AdsWriteOnChange.TcPOU
FUNCTION_BLOCK T_AdsWriteOnChange
VAR
    DataAddress : PVOID;
    DataLength  : UDINT;
    PollTime    : LREAL; // seconds

    AmsNetId            : T_AmsNetID;
    AmsPort             : T_AmsPort;
    SymbolNameToWriteTo : T_Maxstring;

    StructureMonitor       : T_StructureMonitor;
    ValueMonitor           : T_ValueMonitorEx;
    OnTimer_Poll           : T_OnTimer(PresetTime := 0.0);
    OnTimer_DisableOnError : T_OnTimer(PresetTime := 30.0);
    AdsWriteBySymbolName   : T_AdsWriteBySymbolName;
    CommsError             : BOOL;
    pBuffer                : POINTER TO BYTE;
END_VAR

IF DataAddress = 0 OR DataLength = 0 OR pBuffer = 0 THEN
    RETURN;
END_IF

// Disable comms for 30s on comms error to avoid flooding ADS...
IF AdsWriteBySymbolName.Execution.Error THEN
    CommsError := TRUE;
END_IF

IF OnTimer_DisableOnError.Delay(CommsError) THEN
    CommsError := FALSE;
END_IF

// Poll timer:
IF OnTimer_Poll.Delay(AdsWriteBySymbolName.Execution.Ready AND NOT CommsError) THEN

    // Detect any change...
    StructureMonitor.Test(StructureAddress := DataAddress,
                          StructureSize    := DataLength);

    // Write data...
    IF StructureMonitor.Changed THEN
        // Copy data to a buffer - it might have changed before we get round to sending it...
        MEMCPY(destAddr := pBuffer,
               srcAddr  := DataAddress,
               n        := DataLength);

        // send the data...    
        AdsWriteBySymbolName.Execute(AmsNetId         := AmsNetId,
                                     Port             := AmsPort,
                                     SymbolName       := SymbolNameToWriteTo,
                                     WriteDataAddress := pBuffer,
                                     WriteDataLength  := DataLength,
                                     KeepSymbolHandle := TRUE);
    END_IF
END_IF

AdsWriteBySymbolName();

PROPERTY Execution : I_Execution
GET
Execution := AdsWriteBySymbolName.Execution;
END_GET
END_PROPERTY

METHOD FB_exit : BOOL
VAR_INPUT
    bInCopyCode : BOOL; // if TRUE, the exit method is called for exiting an instance that is copied afterwards (online change).
END_VAR
IF NOT bInCopyCode THEN
    __DELETE(pBuffer);
END_IF
END_METHOD

METHOD Initialise
VAR_INPUT
    DataAddress : PVOID;
    DataLength  : UDINT;
    PollTime    : LREAL; // seconds

    AmsNetId            : T_AmsNetID;
    AmsPort             : T_AmsPort;
    SymbolNameToWriteTo : T_Maxstring;
END_VAR
THIS^.DataAddress := DataAddress;
THIS^.DataLength  := DataLength;
THIS^.PollTime    := PollTime;

THIS^.AmsNetId            := AmsNetId;
THIS^.AmsPort             := AmsPort;
THIS^.SymbolNameToWriteTo := SymbolNameToWriteTo;

pBuffer := __NEW(BYTE, DataLength);
END_METHOD

END_FUNCTION_BLOCK
